TYPE stSettings_Skill EXTENDS stSettings_Base :
STRUCT
	
END_STRUCT
END_TYPE

(* stored: Version 1.1.0.1, ProductVersion 3.1.4026.18
   DUT stSettings_Skill: Id {1f54a1c4-096c-4b7e-b281-c442f5aa9d45} *)
